// TIA Portal V17 export
// export: Created 2025-03-13T10:31:24.349857Z, ExportSetting WithDefaults, DisplayName Totally Integrated Automation Portal, DisplayVersion V17 Update 8, DisplayName TIA Portal Openness, DisplayVersion V17 Update 8, DisplayName TIA Portal Version Control Interface, DisplayVersion V17, DisplayName SINAMICS Startdrive Advanced, DisplayVersion V17 SP2, DisplayName SINAMICS Startdrive G110M, G120, G120C, G120D, G120P, G115D, DisplayVersion V17 SP2, DisplayName SINAMICS Startdrive G130, G150, S120, S150, SINAMICS MV, S210, DisplayVersion V17 SP2, DisplayName STEP 7 Professional, DisplayVersion V17 Update 8, DisplayName SINUMERIK ONE STEP 7 Toolbox, DisplayVersion V17 Update 12, DisplayName SINUMERIK 840D sl STEP 7 Toolbox, DisplayVersion V17 Update 12, DisplayName STEP 7 Safety, DisplayVersion V17 Update 6, DisplayName WinCC Advanced, DisplayVersion V17 Update 8
TYPE "SPINDLES_VIBRATIONS"
// stored: IsFailsafeCompliant false
   STRUCT
      VIBRATIONS_RMS_SP1 : Struct   // VIBRATIONS RMS SP1
         VALUE_M_S : Real;
         ERROR : Word;
         WARNING : Real;
         DAMAGE : Real;
         BASE_LINE_M_S : Real;
      END_STRUCT;
      VIBRATIONS_RMS_SP2 : Struct   // VIBRATIONS RMS SP2
         VALUE_M_S : Real;
         ERROR : Word;
         WARNING : Real;
         DAMAGE : Real;
         BASE_LINE_M_S : Real;
      END_STRUCT;
      VIBRATIONS_RMS_SP3 : Struct   // VIBRATIONS RMS SP3
         VALUE_M_S : Real;
         ERROR : Word;
         WARNING : Real;
         DAMAGE : Real;
         BASE_LINE_M_S : Real;
      END_STRUCT;
      VIBRATIONS_RMS_SP4 : Struct   // VIBRATIONS RMS SP4
         VALUE_M_S : Real;
         ERROR : Word;
         WARNING : Real;
         DAMAGE : Real;
         BASE_LINE_M_S : Real;
      END_STRUCT;
      PEAK_TIME_SP1 : Struct   // PEAK TIME SP1
         VALUE_M_S : Real;
         ERROR : Word;
         WARNING : Real;
         DAMAGE : Real;
         BASE_LINE_M_S : Real;
      END_STRUCT;
      PEAK_TIME_SP2 : Struct   // PEAK TIME SP2
         VALUE_M_S : Real;
         ERROR : Word;
         WARNING : Real;
         DAMAGE : Real;
         BASE_LINE_M_S : Real;
      END_STRUCT;
      PEAK_TIME_SP3 : Struct   // PEAK TIME SP3
         VALUE_M_S : Real;
         ERROR : Word;
         WARNING : Real;
         DAMAGE : Real;
         BASE_LINE_M_S : Real;
      END_STRUCT;
      PEAK_TIME_SP4 : Struct   // PEAK TIME SP4
         VALUE_M_S : Real;
         ERROR : Word;
         WARNING : Real;
         DAMAGE : Real;
         BASE_LINE_M_S : Real;
      END_STRUCT;
      VIBRATIONS_RMS_STATE_SP1 : Byte;   // VIBRATIONS RMS STATE SP1
      VIBRATIONS_RMS_STATE_SP2 : Byte;   // VIBRATIONS RMS STATE SP2
      VIBRATIONS_RMS_STATE_SP3 : Byte;   // VIBRATIONS RMS STATE SP3
      VIBRATIONS_RMS_STATE_SP4 : Byte;   // VIBRATIONS RMS STATE SP4
      VIBRATIONS_PEAK_TIME_STATE_SP1 : Byte;   // VIBRATIONS PEAK TIME STATE SP1
      VIBRATIONS_PEAK_TIME_STATE_SP2 : Byte;   // VIBRATIONS PEAK TIME STATE SP2
      VIBRATIONS_PEAK_TIME_STATE_SP3 : Byte;   // VIBRATIONS PEAK TIME STATE SP3
      VIBRATIONS_PEAK_TIME_STATE_SP4 : Byte;   // VIBRATIONS PEAK TIME STATE SP4
      SPARE : Array[0..7] of Byte;
   END_STRUCT;
END_TYPE
